TYPE ST_SoftSettings_PeakshaveBox :
STRUCT
	PeakshaveMode						: ePeakshaveMode;
	setpointTimeslot1					: ST_peakshave_setpoints;
	setpointTimeslot2					: ST_peakshave_setpoints;
	
	b_BreakerControl					: BOOL; // requires fb of mains breaker.
	b_ReverseCTDirection				: BOOL;
	ui_CTrange							: UINT;
	r_VTratio							: REAL := 1; // 1: 1 to 1 (400V), 2: 2 to 1 (800V), ex. 10kV = 25 etc.
END_STRUCT
END_TYPE

(* stored: Version 1.1.0.1, ProductVersion 3.1.4026.18
   DUT ST_SoftSettings_PeakshaveBox: Id {61b09ff7-206a-487b-890c-11d6d00376dc} *)
